Staubli VAL3: chinese.dtx

public string sCancel = "Cancel"
public string sCircular = "Circular"
string sEvtMsg
public string sLinear = "Linear"
public string sListOfMessage[73]
  [0] = "Conveyor calibration utility"
  [1] = "Define conveyor geometry"
  [2] = "Define vision frame"
  [3] = "Define scale factor"
  [4] = "Conveyor overview"
  [5] = "Setup general parameter"
  [6] = "Setup encoder parameter"
  [7] = "Setup detection parameter"
  [8] = "Setup conveyor parameter"
  [9] = "Conveyor Lib."
  [10] = "Encoder Lib."
  [11] = "Detection Lib."
  [12] = "Conveyor type"
  [13] = "Load calibration file"
  [14] = "Conveyor library *\../* is not started, the frame *\../* could not be computed."
  [15] = "Saving successfull"
  [16] = "The library *\../* is going to be deleted, are you sure ?"
  [17] = "Deleting existing conveyor file"
  [18] = "Saving conveyor library"
  [19] = "Saving geometry library"
  [20] = "是否需要检测刚定义的传送带库?"
  [21] = "Libary name : "
  [22] = "No message pending"
  [23] = "Do you want to define a custom origine for the conveyor's frame"
  [24] = "Error code * while computing the frame associated with the conveyor."
  [25] = "Error while computing vision frame : *"
  [26] = "The digital output selected for the clockSignal parameter is not valid."
  [27] = "The digital output selected for reporting robot motion through the upstream end of conveyor window is not valid"
  [28] = "The digital output selected for reporting robot motion through the downstream end of conveyor window is not valid"
  [30] = "The conveyor library *\../* could not be loaded because of error code * "
  [31] = "The encoder library *\../* could not be loaded because of error code * "
  [32] = "The detection library *\../* could not be loaded because of error code * "
  [33] = "The geometry library *\../* could not be loaded because of error code * "
  [34] = "Your current conveyor library *\../* is beeing saved. Please wait..."
  [35] = "The existing conveyor library *\../* could not be replaced, error code *"
  [36] = "The conveyor library *\../* could not be saved because of error code *"
  [37] = "The geometry library *\../* could not be saved because of error code *"
  [38] = "Wizard>>Couldn't find language file:"
  [40] = "Disable any jog mode"
  [41] = "Disable any jog mode"
  [42] = "Disable the Joint jog mode"
  [43] = "Disable the Frame jog mode"
  [44] = "Disable the Tool jog mode"
  [45] = "Disable the Point jog mode"
  [46] = "Warning, This application requires VAL3 version s7.6.0 or higher"
  [47] = "The valTrack license is not installed or demo period has expired."
  [48] = "Loading your conveyor library *\../* into memory. Please wait..."
  [49] = "Initializing conveyor library"
  [50] = "loading geometry library"
  [51] = "loading encoder library"
  [52] = "loading detection library"
  [53] = "Cannot move to the approach of the current robot position. Please check approach TRSF X=* Y=* Z=*."
  [54] = "Cannot move to the approach of the final destination. Please check approach TRSF X=* Y=* Z=*."
  [55] = "Destination is the out of reach."
  [56] = "Warning: Conveyor not created. Create socket client called 'cognex*', camera's IP address, port 1023, timeout 0. Reload wizard."
  [57] = "Warning: Conveyor not selected. Create socket client called 'cognex*', camera's IP address, port 1023, timeout 0. Reload wizard."
  [58] = "Warning: The output defined as ClkSignal doesn't exist"
  [59] = "欢迎进入传送带库设置程序"
  [60] = "选择或新建一个传送带库"
  [61] = "警告：传送带库无法创建。请先创建一个socket服务器，命名"fromRobot_sk*"，端口号100*。重载程序。"
  [62] = "Warning: Conveyor not selected. Create a socket server called 'fromRobot_sk*', port 100*. Reload wizard."
  [63] = "Warning: Message not sent. The socket sent as a parameter is not working. Bad link or device in error."
  [64] = "Warning: Message not sent. Timeout expired. The other robot is not present on the network."
  [65] = "Warning: Message not sent. Timeout expired. The other robot is not working with the detection library 'Socket'."
  [66] = "Warning: Message sent, but the server from the other robot didn't acknowledge reception before expiration of timeout."
  [67] = "VALTRACK"
  [68] = "Warning: Conveyor not created. Edit library Tracking\io\sockets, add to the array of the variable skCognex the index *"
  [69] = "Warning: Conveyor not created. Edit library Tracking\io\sockets, add to the array of the variable skFromRobot the index *"
  [70] = "Warning: Conveyor not selected. Edit library Tracking\io\sockets, add to the array of the variable skCognex the index *"
  [71] = "Warning: Conveyor not selected. Edit library Tracking\io\sockets, add to the array of the variable skFromRobot the index *"
  [72] = "确定取消吗?"
public string sMenu[60]
  [0] = "; ; ; OK ; ; 取消"
  [1] = "; ; ; OK"
  [4] = "上步 未做 选择 ; 平均 ; 下步 取消"
  [5] = "上步 ; ; 调整 ; ; 下步 取消"
  [6] = "上步 记录 移动 ; ; ; 下步 取消"
  [7] = "上步 记录 ; ; ; ; 下步 取消"
  [8] = "上步 ; ; ; ; ; ; 取消"
  [9] = "; ; ; ; ; ; 下步 取消"
  [10] = "; 新建 复制 选择 ; 删除  ; 退出"
  [11] = "; 新建 ; ; ; ; ; 退出"
  [12] = "; ; ; 选择 ; ; ; 取消"
  [13] = "上步 ; ; 选择 ; ; ; 取消"
  [14] = "; 记录 移动 ; ; 帮助 下步 取消"
  [15] = "; 记录 ; ; ; 帮助 下步 取消"
  [16] = "上步 记录 移动 ; ; 帮助 下步 取消"
  [17] = "上步 记录 ; ; ; 帮助 下步 取消"
  [18] = "上步 ; ; ; ; ; 下步 取消"
  [19] = "上步 新建 ; 选择 ; ; ; 取消"
  [20] = "上步 新建 ; ; ; ; ; 取消"
  [21] = "; ; 是 ; ; ; 否"
  [22] = "; ; 是 ; ; ;  否 取消"
  [23] = "; 锁定 ; ; ; ; 下步 取消"
  [50] = "F1: 定义编码器比例因数"
  [51] = "F2: 传送带库坐标系"
  [52] = "F3: 定义传感器距离"
  [53] = "F4: 传送带库诊断"
  [54] = "F5: 完整的校准"
  [55] = "F8: 退出"
public string sNONE = "none"
public string sNOTDEFINED = "Not defined"
public string sNo = "No"
public string sOptionTitle
public string sYes = "Yes"
public trsf trTrsf[4]
public mdesc mNomSpeed = {blend=off}
